{attribute addProperty BoxType "KL6904"}
{attribute addProperty Id "Channel_1Channel_CC0B3E2900"}
{attribute addProperty CRC "388789281"}
{attribute addProperty SizeInBites "0"}
{attribute addProperty SizeInBytes "0"}
TYPE KL6904_172C7421 :
STRUCT
	{attribute addProperty Name "Channel_1"}
	Channel_1 : Channel_CC0B3E29;
END_STRUCT
END_TYPE

(* stored: Version 1.2.0.0, ProductVersion 3.1.4024.9
   DUT KL6904_172C7421: Id {5dc3f943-2eb4-4e5e-ad1c-5adc2b8c72c3} *)
